SPLINE
SPL {X  -165.650, Y  +484.445, Z    +0.000, E1   +32.277, E3 +500064.677}
SPL {X  -165.650, Y  +481.524, Z    +0.000, E1   +31.089, E3 +500082.127}
SPL {X  -165.650, Y  +478.014, Z    +0.000, E1   +30.826, E3 +500095.735}
SPL {X  -165.650, Y  +474.473, Z    +0.000, E1   +30.943, E3 +500107.059}
SPL {X  -165.650, Y  +471.826, Z    +0.000, E1   +30.770, E3 +500117.243}
SPL {X  -165.650, Y  +467.753, Z    +0.000, E1   +30.878, E3 +500130.616}
SPL {X  -165.650, Y  +463.837, Z    +0.000, E1   +30.924, E3 +500143.550}
SPL {X  -165.650, Y  +461.106, Z    +0.000, E1   +30.916, E3 +500152.937}
SPL {X  -165.650, Y  +458.435, Z    +0.000, E1   +30.759, E3 +500163.145}
SPL {X  -165.650, Y  +454.220, Z    +0.000, E1   +30.954, E3 +500176.378}
SPL {X  -165.650, Y  +450.433, Z    +0.000, E1   +30.789, E3 +500190.343}
SPL {X  -165.650, Y  +447.097, Z    +0.000, E1   +30.843, E3 +500201.392}
SPL {X  -165.650, Y  +443.673, Z    +0.000, E1   +30.907, E3 +500212.699}
SPL {X  -165.650, Y  +440.976, Z    +0.000, E1   +30.719, E3 +500223.156}
SPL {X  -165.650, Y  +436.324, Z    +0.000, E1   +30.994, E3 +500237.442}
SPL {X  -165.650, Y  +432.765, Z    +0.000, E1   +30.831, E3 +500250.442}
SPL {X  -165.650, Y  +429.309, Z    +0.000, E1   +30.920, E3 +500261.783}
SPL {X  -165.650, Y  +424.918, Z    +0.000, E1   +30.862, E3 +500277.240}
SPL {X  -165.650, Y  +421.437, Z    +0.000, E1   +30.833, E3 +500289.209}
SPL {X  -165.650, Y  +417.366, Z    +0.000, E1   +30.879, E3 +500303.049}
SPL {X  -165.650, Y  +413.181, Z    +0.000, E1   +30.815, E3 +500317.647}
SPL {X  -165.650, Y  +408.547, Z    +0.000, E1   +30.964, E3 +500332.649}
SPL {X  -165.650, Y  +403.421, Z    +0.000, E1   +30.863, E3 +500350.867}
SPL {X  -165.650, Y  +398.147, Z    +0.000, E1   +30.902, E3 +500368.628}
SPL {X  -165.650, Y  +394.694, Z    +0.000, E1   +30.805, E3 +500380.936}
SPL {X  -165.650, Y  +391.522, Z    +0.000, E1   +30.837, E3 +500391.617}
SPL {X  -165.650, Y  +387.533, Z    +0.000, E1   +30.858, E3 +500405.243}
SPL {X  -165.650, Y  +383.627, Z    +0.000, E1   +30.885, E3 +500418.303}
SPL {X  -165.650, Y  +379.886, Z    +0.000, E1   +30.887, E3 +500431.192}
SPL {X  -165.614, Y  +375.058, Z    +0.000, E1   +30.905, E3 +500447.645}
SPL {X  -165.492, Y  +371.263, Z    +0.000, E1   +30.913, E3 +500460.359}
SPL {X  -165.379, Y  +369.027, Z    +0.000, E1   +30.727, E3 +500469.297}
SPL {X  -165.167, Y  +365.866, Z    +0.000, E1   +30.741, E3 +500480.071}
SPL {X  -164.892, Y  +362.671, Z    +0.000, E1   +30.830, E3 +500490.395}
SPL {X  -164.570, Y  +359.612, Z    +0.000, E1   +30.773, E3 +500501.208}
SPL {X  -164.104, Y  +355.923, Z    +0.000, E1   +30.626, E3 +500514.924}
SPL {X  -163.573, Y  +352.353, Z    +0.000, E1   +30.451, E3 +500528.189}
SPL {X  -162.476, Y  +346.230, Z    +0.000, E1   +31.677, E3 +500540.770}
SPL {X  -152.976, Y  +314.952, Z    +0.000, E1   +38.607, E3 +500589.735}
SPL {X  -137.967, Y  +286.821, Z    +0.000, E1   +43.969, E3 +500632.956}
ENDSPLINE

SPLINE
SPL {X  -153.316, Y  +315.777, Z    +0.000, E1   +33.140, E3 +500675.584}
SPL {X  -164.446, Y  +358.564, Z    +0.000, E1   +15.149, E3 +500640.795}
SPL {X  -165.510, Y  +371.680, Z    +0.000, E1    +7.684, E3 +500644.850}
SPL {X  -165.628, Y  +375.818, Z    +0.000, E1    +5.016, E3 +500652.780}
SPL {X  -165.650, Y  +383.362, Z    +0.000, E1    +0.177, E3 +500633.813}
SPL {X  -165.650, Y  +383.923, Z    +0.000, E1    -0.215, E3 +500646.971}
SPL {X  -165.650, Y  +388.083, Z    +0.000, E1    -3.355, E3 +500645.834}
SPL {X  -165.650, Y  +395.510, Z    +0.000, E1    -9.810, E3 +500641.960}
SPL {X  -165.650, Y  +403.066, Z    +0.000, E1   -17.886, E3 +500634.793}
SPL {X  -165.650, Y  +414.811, Z    +0.000, E1   -28.314, E3 +500636.275}
SPL {X  -165.650, Y  +423.479, Z    +0.000, E1   -29.012, E3 +500660.203}
SPL {X  -165.650, Y  +435.050, Z    +0.000, E1   -34.610, E3 +500668.538}
SPL {X  -165.650, Y  +446.725, Z    +0.000, E1   -39.593, E3 +500674.799}
SPL {X  -165.650, Y  +462.890, Z    +0.000, E1   -40.484, E3 +500705.975}
ENDSPLINE

SPLINE
SPL {X  -165.650, Y  +446.920, Z    +0.000, E1   -31.238, E3 +500718.301}
ENDSPLINE

SPLINE
SPL {X  -165.650, Y  +447.935, Z    +0.000, E1   -30.213, E3 +500728.589}
SPL {X  -165.650, Y  +451.020, Z    +0.000, E1   -30.224, E3 +500739.409}
SPL {X  -165.650, Y  +454.519, Z    +0.000, E1   -30.374, E3 +500750.592}
SPL {X  -165.650, Y  +457.429, Z    +0.000, E1   -30.029, E3 +500763.293}
SPL {X  -165.650, Y  +461.678, Z    +0.000, E1   -30.426, E3 +500775.418}
SPL {X  -165.650, Y  +463.853, Z    +0.000, E1   -30.103, E3 +500785.258}
SPL {X  -165.650, Y  +468.397, Z    +0.000, E1   -30.302, E3 +500800.061}
SPL {X  -165.650, Y  +472.566, Z    +0.000, E1   -30.124, E3 +500815.771}
SPL {X  -165.650, Y  +475.265, Z    +0.000, E1   -30.034, E3 +500825.808}
SPL {X  -165.650, Y  +477.862, Z    +0.000, E1   -30.319, E3 +500833.000}
SPL {X  -165.650, Y  +481.042, Z    +0.000, E1   -30.192, E3 +500845.260}
SPL {X  -165.650, Y  +485.236, Z    +0.000, E1   -30.294, E3 +500859.116}
SPL {X  -165.650, Y  +488.041, Z    +0.000, E1   -30.253, E3 +500869.237}
SPL {X  -165.650, Y  +491.281, Z    +0.000, E1   -30.148, E3 +500881.375}
SPL {X  -165.650, Y  +495.051, Z    +0.000, E1   -30.213, E3 +500894.184}
SPL {X  -165.650, Y  +499.546, Z    +0.000, E1   -30.283, E3 +500909.627}
SPL {X  -165.650, Y  +503.544, Z    +0.000, E1   -30.247, E3 +500923.695}
SPL {X  -165.650, Y  +506.344, Z    +0.000, E1   -30.129, E3 +500934.364}
SPL {X  -165.650, Y  +509.866, Z    +0.000, E1   -30.236, E3 +500946.033}
SPL {X  -165.650, Y  +513.685, Z    +0.000, E1   -30.234, E3 +500959.529}
SPL {X  -165.650, Y  +517.919, Z    +0.000, E1   -30.227, E3 +500974.436}
SPL {X  -165.650, Y  +521.521, Z    +0.000, E1   -30.210, E3 +500987.111}
SPL {X  -165.650, Y  +525.344, Z    +0.000, E1   -30.269, E3 +501000.217}
SPL {X  -165.650, Y  +528.152, Z    +0.000, E1   -29.991, E3 +501011.858}
SPL {X  -165.650, Y  +531.783, Z    +0.000, E1   -30.416, E3 +501021.751}
SPL {X  -165.650, Y  +534.115, Z    +0.000, E1   -30.089, E3 +501032.133}
SPL {X  -165.650, Y  +537.522, Z    +0.000, E1   -30.251, E3 +501043.047}
SPL {X  -165.650, Y  +540.621, Z    +0.000, E1   -30.014, E3 +501055.608}
SPL {X  -165.650, Y  +544.944, Z    +0.000, E1   -30.447, E3 +501067.808}
SPL {X  -165.650, Y  +547.199, Z    +0.000, E1   -30.132, E3 +501077.782}
SPL {X  -165.650, Y  +550.512, Z    +0.000, E1   -30.197, E3 +501089.107}
SPL {X  -165.650, Y  +553.852, Z    +0.000, E1   -30.156, E3 +501101.048}
SPL {X  -165.650, Y  +557.277, Z    +0.000, E1   -30.150, E3 +501113.223}
SPL {X  -165.650, Y  +561.168, Z    +0.000, E1   -30.194, E3 +501126.604}
SPL {X  -165.650, Y  +565.528, Z    +0.000, E1   -30.192, E3 +501142.087}
SPL {X  -165.650, Y  +570.048, Z    +0.000, E1   -30.238, E3 +501157.518}
SPL {X  -165.650, Y  +573.110, Z    +0.000, E1   -30.057, E3 +501169.503}
SPL {X  -165.650, Y  +577.587, Z    +0.000, E1   -30.270, E3 +501183.942}
SPL {X  -165.650, Y  +581.190, Z    +0.000, E1   -30.107, E3 +501197.581}
SPL {X  -165.650, Y  +585.053, Z    +0.000, E1   -30.090, E3 +501211.451}
ENDSPLINE

SPLINE
SPL {X  -165.650, Y  +484.445, Z    +0.000, E1   +32.277, E3 +501228.856}
SPL {X  -165.650, Y  +481.524, Z    +0.000, E1   +31.089, E3 +501246.306}
SPL {X  -165.650, Y  +478.014, Z    +0.000, E1   +30.826, E3 +501259.914}
SPL {X  -165.650, Y  +474.473, Z    +0.000, E1   +30.943, E3 +501271.238}
SPL {X  -165.650, Y  +471.826, Z    +0.000, E1   +30.770, E3 +501281.422}
SPL {X  -165.650, Y  +467.753, Z    +0.000, E1   +30.878, E3 +501294.795}
SPL {X  -165.650, Y  +463.837, Z    +0.000, E1   +30.924, E3 +501307.729}
SPL {X  -165.650, Y  +461.106, Z    +0.000, E1   +30.916, E3 +501317.116}
SPL {X  -165.650, Y  +458.435, Z    +0.000, E1   +30.759, E3 +501327.324}
SPL {X  -165.650, Y  +454.220, Z    +0.000, E1   +30.954, E3 +501340.557}
SPL {X  -165.650, Y  +450.433, Z    +0.000, E1   +30.789, E3 +501354.522}
SPL {X  -165.650, Y  +447.097, Z    +0.000, E1   +30.843, E3 +501365.571}
SPL {X  -165.650, Y  +443.673, Z    +0.000, E1   +30.907, E3 +501376.878}
SPL {X  -165.650, Y  +440.976, Z    +0.000, E1   +30.719, E3 +501387.335}
SPL {X  -165.650, Y  +436.324, Z    +0.000, E1   +30.994, E3 +501401.621}
SPL {X  -165.650, Y  +432.765, Z    +0.000, E1   +30.831, E3 +501414.621}
SPL {X  -165.650, Y  +429.309, Z    +0.000, E1   +30.920, E3 +501425.962}
SPL {X  -165.650, Y  +424.918, Z    +0.000, E1   +30.862, E3 +501441.419}
SPL {X  -165.650, Y  +421.437, Z    +0.000, E1   +30.833, E3 +501453.388}
SPL {X  -165.650, Y  +418.489, Z    +0.000, E1   +30.835, E3 +501463.504}
SPL {X  -165.650, Y  +414.127, Z    +0.000, E1   +30.869, E3 +501478.413}
SPL {X  -165.650, Y  +408.547, Z    +0.000, E1   +30.964, E3 +501496.829}
SPL {X  -165.650, Y  +405.433, Z    +0.000, E1   +30.730, E3 +501508.806}
SPL {X  -165.650, Y  +401.473, Z    +0.000, E1   +30.933, E3 +501521.254}
SPL {X  -165.650, Y  +396.018, Z    +0.000, E1   +30.861, E3 +501540.439}
SPL {X  -165.650, Y  +391.522, Z    +0.000, E1   +30.837, E3 +501555.796}
SPL {X  -165.650, Y  +387.533, Z    +0.000, E1   +30.858, E3 +501569.422}
SPL {X  -165.650, Y  +383.627, Z    +0.000, E1   +30.885, E3 +501582.483}
SPL {X  -165.650, Y  +380.752, Z    +0.000, E1   +30.927, E3 +501591.996}
SPL {X  -165.648, Y  +377.739, Z    +0.000, E1   +30.835, E3 +501603.006}
SPL {X  -165.594, Y  +374.183, Z    +0.000, E1   +30.878, E3 +501614.843}
SPL {X  -165.429, Y  +369.945, Z    +0.000, E1   +30.850, E3 +501629.718}
SPL {X  -165.167, Y  +365.866, Z    +0.000, E1   +30.741, E3 +501644.250}
SPL {X  -164.892, Y  +362.671, Z    +0.000, E1   +30.830, E3 +501654.574}
SPL {X  -164.570, Y  +359.612, Z    +0.000, E1   +30.773, E3 +501665.387}
SPL {X  -164.104, Y  +355.923, Z    +0.000, E1   +30.626, E3 +501679.104}
SPL {X  -163.573, Y  +352.353, Z    +0.000, E1   +30.451, E3 +501692.368}
SPL {X  -162.976, Y  +348.856, Z    +0.000, E1   +30.757, E3 +501702.292}
SPL {X  -161.497, Y  +341.640, Z    +0.000, E1   +33.276, E3 +501709.570}
SPL {X  -152.976, Y  +314.952, Z    +0.000, E1   +38.607, E3 +501753.914}
SPL {X  -137.967, Y  +286.821, Z    +0.000, E1   +43.969, E3 +501797.135}
ENDSPLINE

SPLINE
SPL {X  -149.143, Y  +306.414, Z    +0.000, E1   +36.361, E3 +501848.268}
SPL {X  -164.268, Y  +357.145, Z    +0.000, E1   +15.880, E3 +501806.027}
SPL {X  -165.510, Y  +371.680, Z    +0.000, E1    +7.684, E3 +501809.029}
SPL {X  -165.628, Y  +375.818, Z    +0.000, E1    +5.016, E3 +501816.959}
SPL {X  -165.650, Y  +383.362, Z    +0.000, E1    +0.177, E3 +501797.992}
SPL {X  -165.650, Y  +383.923, Z    +0.000, E1    -0.215, E3 +501811.150}
SPL {X  -165.650, Y  +388.083, Z    +0.000, E1    -3.355, E3 +501810.013}
SPL {X  -165.650, Y  +395.510, Z    +0.000, E1    -9.810, E3 +501806.139}
SPL {X  -165.650, Y  +403.066, Z    +0.000, E1   -17.886, E3 +501798.973}
SPL {X  -165.650, Y  +416.345, Z    +0.000, E1   -29.511, E3 +501800.715}
SPL {X  -165.650, Y  +422.331, Z    +0.000, E1   -27.760, E3 +501826.214}
SPL {X  -165.650, Y  +441.276, Z    +0.000, E1   -37.343, E3 +501836.071}
SPL {X  -165.650, Y  +462.890, Z    +0.000, E1   -40.484, E3 +501870.154}
ENDSPLINE

SPLINE
SPL {X  -165.650, Y  +446.920, Z    +0.000, E1   -31.238, E3 +501882.480}
ENDSPLINE

SPLINE
SPL {X  -165.650, Y  +447.935, Z    +0.000, E1   -30.213, E3 +501892.768}
SPL {X  -165.650, Y  +451.020, Z    +0.000, E1   -30.224, E3 +501903.588}
SPL {X  -165.650, Y  +454.519, Z    +0.000, E1   -30.374, E3 +501914.771}
SPL {X  -165.650, Y  +457.429, Z    +0.000, E1   -30.029, E3 +501927.473}
SPL {X  -165.650, Y  +461.678, Z    +0.000, E1   -30.426, E3 +501939.597}
SPL {X  -165.650, Y  +463.853, Z    +0.000, E1   -30.103, E3 +501949.437}
SPL {X  -165.650, Y  +468.397, Z    +0.000, E1   -30.302, E3 +501964.241}
SPL {X  -165.650, Y  +472.566, Z    +0.000, E1   -30.124, E3 +501979.950}
SPL {X  -165.650, Y  +476.540, Z    +0.000, E1   -30.193, E3 +501993.494}
SPL {X  -165.650, Y  +481.042, Z    +0.000, E1   -30.192, E3 +502009.439}
SPL {X  -165.650, Y  +485.236, Z    +0.000, E1   -30.294, E3 +502023.295}
SPL {X  -165.650, Y  +489.057, Z    +0.000, E1   -30.341, E3 +502036.501}
SPL {X  -165.650, Y  +491.647, Z    +0.000, E1   -29.894, E3 +502048.434}
SPL {X  -165.650, Y  +495.051, Z    +0.000, E1   -30.213, E3 +502058.363}
SPL {X  -165.650, Y  +498.418, Z    +0.000, E1   -30.282, E3 +502069.656}
SPL {X  -165.650, Y  +502.421, Z    +0.000, E1   -30.263, E3 +502084.013}
SPL {X  -165.650, Y  +506.344, Z    +0.000, E1   -30.129, E3 +502098.543}
SPL {X  -165.650, Y  +509.866, Z    +0.000, E1   -30.236, E3 +502110.212}
SPL {X  -165.650, Y  +513.685, Z    +0.000, E1   -30.234, E3 +502123.709}
SPL {X  -165.650, Y  +517.919, Z    +0.000, E1   -30.227, E3 +502138.615}
SPL {X  -165.650, Y  +521.521, Z    +0.000, E1   -30.210, E3 +502151.290}
SPL {X  -165.650, Y  +525.344, Z    +0.000, E1   -30.269, E3 +502164.396}
SPL {X  -165.650, Y  +528.152, Z    +0.000, E1   -29.991, E3 +502176.037}
SPL {X  -165.650, Y  +531.783, Z    +0.000, E1   -30.416, E3 +502185.930}
SPL {X  -165.650, Y  +534.115, Z    +0.000, E1   -30.089, E3 +502196.312}
SPL {X  -165.650, Y  +537.522, Z    +0.000, E1   -30.251, E3 +502207.227}
SPL {X  -165.650, Y  +540.621, Z    +0.000, E1   -30.014, E3 +502219.787}
SPL {X  -165.650, Y  +544.944, Z    +0.000, E1   -30.447, E3 +502231.987}
SPL {X  -165.650, Y  +548.549, Z    +0.000, E1   -30.216, E3 +502246.311}
SPL {X  -165.650, Y  +553.092, Z    +0.000, E1   -30.157, E3 +502262.653}
SPL {X  -165.650, Y  +556.274, Z    +0.000, E1   -30.127, E3 +502273.908}
SPL {X  -165.650, Y  +560.243, Z    +0.000, E1   -30.214, E3 +502287.574}
SPL {X  -165.650, Y  +565.528, Z    +0.000, E1   -30.192, E3 +502306.266}
SPL {X  -165.650, Y  +570.048, Z    +0.000, E1   -30.238, E3 +502321.697}
SPL {X  -165.650, Y  +573.110, Z    +0.000, E1   -30.057, E3 +502333.682}
SPL {X  -165.650, Y  +577.587, Z    +0.000, E1   -30.270, E3 +502348.121}
SPL {X  -165.650, Y  +581.190, Z    +0.000, E1   -30.107, E3 +502361.760}
SPL {X  -165.650, Y  +585.053, Z    +0.000, E1   -30.090, E3 +502375.631}
ENDSPLINE

SPLINE
SPL {X  -165.650, Y  +484.445, Z    +0.000, E1   +32.277, E3 +502393.035}
SPL {X  -165.650, Y  +481.524, Z    +0.000, E1   +31.089, E3 +502410.486}
SPL {X  -165.650, Y  +478.014, Z    +0.000, E1   +30.826, E3 +502424.093}
SPL {X  -165.650, Y  +474.473, Z    +0.000, E1   +30.943, E3 +502435.418}
SPL {X  -165.650, Y  +471.826, Z    +0.000, E1   +30.770, E3 +502445.601}
SPL {X  -165.650, Y  +467.753, Z    +0.000, E1   +30.878, E3 +502458.974}
SPL {X  -165.650, Y  +463.837, Z    +0.000, E1   +30.924, E3 +502471.908}
SPL {X  -165.650, Y  +461.106, Z    +0.000, E1   +30.916, E3 +502481.295}
SPL {X  -165.650, Y  +458.435, Z    +0.000, E1   +30.759, E3 +502491.503}
SPL {X  -165.650, Y  +454.220, Z    +0.000, E1   +30.954, E3 +502504.736}
SPL {X  -165.650, Y  +450.433, Z    +0.000, E1   +30.789, E3 +502518.701}
SPL {X  -165.650, Y  +447.097, Z    +0.000, E1   +30.843, E3 +502529.750}
SPL {X  -165.650, Y  +443.673, Z    +0.000, E1   +30.907, E3 +502541.057}
SPL {X  -165.650, Y  +440.976, Z    +0.000, E1   +30.719, E3 +502551.514}
SPL {X  -165.650, Y  +436.324, Z    +0.000, E1   +30.994, E3 +502565.800}
SPL {X  -165.650, Y  +432.765, Z    +0.000, E1   +30.831, E3 +502578.800}
SPL {X  -165.650, Y  +429.309, Z    +0.000, E1   +30.920, E3 +502590.141}
SPL {X  -165.650, Y  +424.918, Z    +0.000, E1   +30.862, E3 +502605.598}
SPL {X  -165.650, Y  +421.437, Z    +0.000, E1   +30.833, E3 +502617.567}
SPL {X  -165.650, Y  +417.366, Z    +0.000, E1   +30.879, E3 +502631.407}
SPL {X  -165.650, Y  +413.181, Z    +0.000, E1   +30.815, E3 +502646.005}
SPL {X  -165.650, Y  +408.547, Z    +0.000, E1   +30.964, E3 +502661.008}
SPL {X  -165.650, Y  +403.421, Z    +0.000, E1   +30.863, E3 +502679.225}
SPL {X  -165.650, Y  +398.147, Z    +0.000, E1   +30.902, E3 +502696.986}
SPL {X  -165.650, Y  +394.694, Z    +0.000, E1   +30.805, E3 +502709.294}
SPL {X  -165.650, Y  +391.522, Z    +0.000, E1   +30.837, E3 +502719.975}
SPL {X  -165.650, Y  +387.533, Z    +0.000, E1   +30.858, E3 +502733.601}
SPL {X  -165.650, Y  +383.627, Z    +0.000, E1   +30.885, E3 +502746.662}
SPL {X  -165.650, Y  +379.886, Z    +0.000, E1   +30.887, E3 +502759.550}
SPL {X  -165.614, Y  +375.058, Z    +0.000, E1   +30.905, E3 +502776.003}
SPL {X  -165.492, Y  +371.263, Z    +0.000, E1   +30.913, E3 +502788.717}
SPL {X  -165.379, Y  +369.027, Z    +0.000, E1   +30.727, E3 +502797.655}
SPL {X  -165.167, Y  +365.866, Z    +0.000, E1   +30.741, E3 +502808.429}
SPL {X  -164.892, Y  +362.671, Z    +0.000, E1   +30.830, E3 +502818.754}
SPL {X  -164.570, Y  +359.612, Z    +0.000, E1   +30.773, E3 +502829.566}
SPL {X  -164.104, Y  +355.923, Z    +0.000, E1   +30.626, E3 +502843.283}
SPL {X  -163.573, Y  +352.353, Z    +0.000, E1   +30.451, E3 +502856.547}
SPL {X  -162.476, Y  +346.230, Z    +0.000, E1   +31.677, E3 +502869.128}
SPL {X  -152.976, Y  +314.952, Z    +0.000, E1   +38.607, E3 +502918.093}
SPL {X  -137.967, Y  +286.821, Z    +0.000, E1   +43.969, E3 +502961.315}
ENDSPLINE

SPLINE
SPL {X  -153.316, Y  +315.777, Z    +0.000, E1   +33.140, E3 +503003.942}
SPL {X  -164.446, Y  +358.564, Z    +0.000, E1   +15.149, E3 +502969.153}
SPL {X  -165.379, Y  +369.025, Z    +0.000, E1    +9.158, E3 +502974.878}
SPL {X  -165.612, Y  +374.969, Z    +0.000, E1    +5.630, E3 +502977.553}
SPL {X  -165.650, Y  +383.362, Z    +0.000, E1    +0.177, E3 +502962.172}
SPL {X  -165.650, Y  +383.923, Z    +0.000, E1    -0.215, E3 +502975.329}
SPL {X  -165.650, Y  +388.083, Z    +0.000, E1    -3.355, E3 +502974.192}
SPL {X  -165.650, Y  +395.510, Z    +0.000, E1    -9.810, E3 +502970.318}
SPL {X  -165.650, Y  +403.066, Z    +0.000, E1   -17.886, E3 +502963.152}
SPL {X  -165.650, Y  +414.811, Z    +0.000, E1   -28.314, E3 +502964.633}
SPL {X  -165.650, Y  +423.479, Z    +0.000, E1   -29.012, E3 +502988.562}
SPL {X  -165.650, Y  +441.276, Z    +0.000, E1   -37.343, E3 +503000.250}
SPL {X  -165.650, Y  +462.890, Z    +0.000, E1   -40.484, E3 +503034.333}
ENDSPLINE

SPLINE
SPL {X  -165.650, Y  +446.920, Z    +0.000, E1   -31.238, E3 +503046.659}
ENDSPLINE

SPLINE
SPL {X  -165.650, Y  +447.935, Z    +0.000, E1   -30.213, E3 +503056.947}
SPL {X  -165.650, Y  +451.020, Z    +0.000, E1   -30.224, E3 +503067.768}
SPL {X  -165.650, Y  +454.519, Z    +0.000, E1   -30.374, E3 +503078.950}
SPL {X  -165.650, Y  +457.429, Z    +0.000, E1   -30.029, E3 +503091.652}
SPL {X  -165.650, Y  +461.678, Z    +0.000, E1   -30.426, E3 +503103.776}
SPL {X  -165.650, Y  +463.853, Z    +0.000, E1   -30.103, E3 +503113.616}
SPL {X  -165.650, Y  +468.397, Z    +0.000, E1   -30.302, E3 +503128.420}
SPL {X  -165.650, Y  +472.566, Z    +0.000, E1   -30.124, E3 +503144.129}
SPL {X  -165.650, Y  +476.540, Z    +0.000, E1   -30.193, E3 +503157.673}
SPL {X  -165.650, Y  +481.042, Z    +0.000, E1   -30.192, E3 +503173.618}
SPL {X  -165.650, Y  +485.236, Z    +0.000, E1   -30.294, E3 +503187.474}
SPL {X  -165.650, Y  +489.057, Z    +0.000, E1   -30.341, E3 +503200.680}
SPL {X  -165.650, Y  +491.647, Z    +0.000, E1   -29.894, E3 +503212.613}
SPL {X  -165.650, Y  +495.051, Z    +0.000, E1   -30.213, E3 +503222.542}
SPL {X  -165.650, Y  +499.546, Z    +0.000, E1   -30.283, E3 +503237.985}
SPL {X  -165.650, Y  +503.544, Z    +0.000, E1   -30.247, E3 +503252.053}
SPL {X  -165.650, Y  +506.344, Z    +0.000, E1   -30.129, E3 +503262.722}
SPL {X  -165.650, Y  +510.660, Z    +0.000, E1   -30.223, E3 +503277.425}
SPL {X  -165.650, Y  +514.670, Z    +0.000, E1   -30.278, E3 +503290.935}
SPL {X  -165.650, Y  +517.919, Z    +0.000, E1   -30.227, E3 +503302.795}
SPL {X  -165.650, Y  +522.822, Z    +0.000, E1   -30.289, E3 +503319.684}
SPL {X  -165.650, Y  +527.393, Z    +0.000, E1   -30.104, E3 +503336.932}
SPL {X  -165.650, Y  +531.783, Z    +0.000, E1   -30.416, E3 +503350.109}
SPL {X  -165.650, Y  +534.115, Z    +0.000, E1   -30.089, E3 +503360.491}
SPL {X  -165.650, Y  +538.363, Z    +0.000, E1   -30.232, E3 +503374.661}
SPL {X  -165.650, Y  +543.650, Z    +0.000, E1   -30.281, E3 +503392.881}
SPL {X  -165.650, Y  +548.549, Z    +0.000, E1   -30.216, E3 +503410.490}
SPL {X  -165.650, Y  +553.092, Z    +0.000, E1   -30.157, E3 +503426.832}
SPL {X  -165.650, Y  +556.274, Z    +0.000, E1   -30.127, E3 +503438.087}
SPL {X  -165.650, Y  +560.243, Z    +0.000, E1   -30.214, E3 +503451.753}
SPL {X  -165.650, Y  +565.528, Z    +0.000, E1   -30.192, E3 +503470.445}
SPL {X  -165.650, Y  +570.048, Z    +0.000, E1   -30.238, E3 +503485.876}
SPL {X  -165.650, Y  +573.110, Z    +0.000, E1   -30.057, E3 +503497.861}
SPL {X  -165.650, Y  +577.587, Z    +0.000, E1   -30.270, E3 +503512.300}
SPL {X  -165.650, Y  +581.190, Z    +0.000, E1   -30.107, E3 +503525.939}
SPL {X  -165.650, Y  +585.053, Z    +0.000, E1   -30.090, E3 +503539.810}
ENDSPLINE

SPLINE
SPL {X  -165.650, Y  +484.445, Z    +0.000, E1   +32.277, E3 +503557.214}
SPL {X  -165.650, Y  +481.524, Z    +0.000, E1   +31.089, E3 +503574.665}
SPL {X  -165.650, Y  +478.014, Z    +0.000, E1   +30.826, E3 +503588.272}
SPL {X  -165.650, Y  +474.473, Z    +0.000, E1   +30.943, E3 +503599.597}
SPL {X  -165.650, Y  +471.826, Z    +0.000, E1   +30.770, E3 +503609.780}
SPL {X  -165.650, Y  +467.753, Z    +0.000, E1   +30.878, E3 +503623.154}
SPL {X  -165.650, Y  +463.837, Z    +0.000, E1   +30.924, E3 +503636.087}
SPL {X  -165.650, Y  +461.106, Z    +0.000, E1   +30.916, E3 +503645.474}
SPL {X  -165.650, Y  +457.156, Z    +0.000, E1   +30.860, E3 +503659.551}
SPL {X  -165.650, Y  +453.156, Z    +0.000, E1   +30.934, E3 +503672.525}
SPL {X  -165.650, Y  +450.433, Z    +0.000, E1   +30.789, E3 +503682.880}
SPL {X  -165.650, Y  +447.097, Z    +0.000, E1   +30.843, E3 +503693.929}
SPL {X  -165.650, Y  +443.673, Z    +0.000, E1   +30.907, E3 +503705.236}
SPL {X  -165.650, Y  +439.486, Z    +0.000, E1   +30.857, E3 +503720.046}
SPL {X  -165.650, Y  +435.146, Z    +0.000, E1   +30.969, E3 +503733.965}
SPL {X  -165.650, Y  +431.607, Z    +0.000, E1   +30.889, E3 +503746.680}
SPL {X  -165.650, Y  +427.340, Z    +0.000, E1   +30.870, E3 +503761.391}
SPL {X  -165.650, Y  +423.901, Z    +0.000, E1   +30.858, E3 +503773.148}
SPL {X  -165.650, Y  +421.437, Z    +0.000, E1   +30.833, E3 +503781.746}
SPL {X  -165.650, Y  +418.489, Z    +0.000, E1   +30.835, E3 +503791.863}
SPL {X  -165.650, Y  +414.127, Z    +0.000, E1   +30.869, E3 +503806.771}
SPL {X  -165.650, Y  +408.547, Z    +0.000, E1   +30.964, E3 +503825.187}
SPL {X  -165.650, Y  +405.433, Z    +0.000, E1   +30.730, E3 +503837.164}
SPL {X  -165.650, Y  +401.473, Z    +0.000, E1   +30.933, E3 +503849.612}
SPL {X  -165.650, Y  +396.018, Z    +0.000, E1   +30.861, E3 +503868.797}
SPL {X  -165.650, Y  +391.522, Z    +0.000, E1   +30.837, E3 +503884.154}
SPL {X  -165.650, Y  +387.533, Z    +0.000, E1   +30.858, E3 +503897.780}
SPL {X  -165.650, Y  +383.627, Z    +0.000, E1   +30.885, E3 +503910.841}
SPL {X  -165.650, Y  +380.752, Z    +0.000, E1   +30.927, E3 +503920.355}
SPL {X  -165.648, Y  +377.739, Z    +0.000, E1   +30.835, E3 +503931.364}
SPL {X  -165.594, Y  +374.183, Z    +0.000, E1   +30.878, E3 +503943.201}
SPL {X  -165.429, Y  +369.945, Z    +0.000, E1   +30.850, E3 +503958.076}
SPL {X  -165.167, Y  +365.866, Z    +0.000, E1   +30.741, E3 +503972.609}
SPL {X  -164.892, Y  +362.671, Z    +0.000, E1   +30.830, E3 +503982.933}
SPL {X  -164.570, Y  +359.612, Z    +0.000, E1   +30.773, E3 +503993.745}
SPL {X  -164.104, Y  +355.923, Z    +0.000, E1   +30.626, E3 +504007.462}
SPL {X  -163.573, Y  +352.353, Z    +0.000, E1   +30.451, E3 +504020.727}
SPL {X  -162.976, Y  +348.856, Z    +0.000, E1   +30.757, E3 +504030.650}
SPL {X  -161.497, Y  +341.640, Z    +0.000, E1   +33.276, E3 +504037.928}
SPL {X  -152.976, Y  +314.952, Z    +0.000, E1   +38.607, E3 +504082.272}
SPL {X  -137.967, Y  +286.821, Z    +0.000, E1   +43.969, E3 +504125.494}
ENDSPLINE

SPLINE
SPL {X  -149.143, Y  +306.414, Z    +0.000, E1   +36.361, E3 +504176.626}
SPL {X  -164.268, Y  +357.145, Z    +0.000, E1   +15.880, E3 +504134.385}
SPL {X  -165.510, Y  +371.680, Z    +0.000, E1    +7.684, E3 +504137.388}
SPL {X  -165.628, Y  +375.818, Z    +0.000, E1    +5.016, E3 +504145.317}
SPL {X  -165.650, Y  +383.362, Z    +0.000, E1    +0.177, E3 +504126.351}
SPL {X  -165.650, Y  +383.923, Z    +0.000, E1    -0.215, E3 +504139.508}
SPL {X  -165.650, Y  +388.083, Z    +0.000, E1    -3.355, E3 +504138.371}
SPL {X  -165.650, Y  +395.510, Z    +0.000, E1    -9.810, E3 +504134.498}
SPL {X  -165.650, Y  +403.066, Z    +0.000, E1   -17.886, E3 +504127.331}
SPL {X  -165.650, Y  +416.345, Z    +0.000, E1   -29.511, E3 +504129.073}
SPL {X  -165.650, Y  +422.331, Z    +0.000, E1   -27.760, E3 +504154.572}
SPL {X  -165.650, Y  +441.276, Z    +0.000, E1   -37.343, E3 +504164.430}
SPL {X  -165.650, Y  +462.890, Z    +0.000, E1   -40.484, E3 +504198.512}
ENDSPLINE

SPLINE
SPL {X  -165.650, Y  +446.920, Z    +0.000, E1   -31.238, E3 +504210.838}
ENDSPLINE

SPLINE
SPL {X  -165.650, Y  +447.935, Z    +0.000, E1   -30.213, E3 +504221.126}
SPL {X  -165.650, Y  +451.020, Z    +0.000, E1   -30.224, E3 +504231.947}
SPL {X  -165.650, Y  +454.519, Z    +0.000, E1   -30.374, E3 +504243.129}
SPL {X  -165.650, Y  +457.429, Z    +0.000, E1   -30.029, E3 +504255.831}
SPL {X  -165.650, Y  +461.678, Z    +0.000, E1   -30.426, E3 +504267.955}
SPL {X  -165.650, Y  +463.853, Z    +0.000, E1   -30.103, E3 +504277.795}
SPL {X  -165.650, Y  +468.397, Z    +0.000, E1   -30.302, E3 +504292.599}
SPL {X  -165.650, Y  +472.566, Z    +0.000, E1   -30.124, E3 +504308.308}
SPL {X  -165.650, Y  +476.540, Z    +0.000, E1   -30.193, E3 +504321.852}
SPL {X  -165.650, Y  +481.042, Z    +0.000, E1   -30.192, E3 +504337.797}
SPL {X  -165.650, Y  +485.236, Z    +0.000, E1   -30.294, E3 +504351.653}
SPL {X  -165.650, Y  +489.057, Z    +0.000, E1   -30.341, E3 +504364.859}
SPL {X  -165.650, Y  +491.647, Z    +0.000, E1   -29.894, E3 +504376.792}
SPL {X  -165.650, Y  +495.051, Z    +0.000, E1   -30.213, E3 +504386.721}
SPL {X  -165.650, Y  +498.418, Z    +0.000, E1   -30.282, E3 +504398.014}
SPL {X  -165.650, Y  +502.421, Z    +0.000, E1   -30.263, E3 +504412.371}
SPL {X  -165.650, Y  +506.344, Z    +0.000, E1   -30.129, E3 +504426.901}
SPL {X  -165.650, Y  +509.866, Z    +0.000, E1   -30.236, E3 +504438.570}
SPL {X  -165.650, Y  +513.685, Z    +0.000, E1   -30.234, E3 +504452.067}
SPL {X  -165.650, Y  +517.919, Z    +0.000, E1   -30.227, E3 +504466.974}
SPL {X  -165.650, Y  +521.521, Z    +0.000, E1   -30.210, E3 +504479.648}
SPL {X  -165.650, Y  +525.344, Z    +0.000, E1   -30.269, E3 +504492.755}
SPL {X  -165.650, Y  +528.152, Z    +0.000, E1   -29.991, E3 +504504.396}
SPL {X  -165.650, Y  +531.783, Z    +0.000, E1   -30.416, E3 +504514.288}
SPL {X  -165.650, Y  +534.115, Z    +0.000, E1   -30.089, E3 +504524.670}
SPL {X  -165.650, Y  +537.522, Z    +0.000, E1   -30.251, E3 +504535.585}
SPL {X  -165.650, Y  +540.621, Z    +0.000, E1   -30.014, E3 +504548.146}
SPL {X  -165.650, Y  +544.944, Z    +0.000, E1   -30.447, E3 +504560.345}
SPL {X  -165.650, Y  +548.549, Z    +0.000, E1   -30.216, E3 +504574.669}
SPL {X  -165.650, Y  +553.092, Z    +0.000, E1   -30.157, E3 +504591.011}
SPL {X  -165.650, Y  +556.274, Z    +0.000, E1   -30.127, E3 +504602.266}
SPL {X  -165.650, Y  +560.243, Z    +0.000, E1   -30.214, E3 +504615.932}
SPL {X  -165.650, Y  +565.528, Z    +0.000, E1   -30.192, E3 +504634.624}
SPL {X  -165.650, Y  +570.048, Z    +0.000, E1   -30.238, E3 +504650.055}
SPL {X  -165.650, Y  +573.110, Z    +0.000, E1   -30.057, E3 +504662.040}
SPL {X  -165.650, Y  +577.587, Z    +0.000, E1   -30.270, E3 +504676.479}
SPL {X  -165.650, Y  +581.190, Z    +0.000, E1   -30.107, E3 +504690.119}
SPL {X  -165.650, Y  +585.053, Z    +0.000, E1   -30.090, E3 +504703.989}
ENDSPLINE

SPLINE
SPL {X  -165.650, Y  +484.445, Z    +0.000, E1   +32.277, E3 +504721.393}
SPL {X  -165.650, Y  +481.524, Z    +0.000, E1   +31.089, E3 +504738.844}
SPL {X  -165.650, Y  +478.014, Z    +0.000, E1   +30.826, E3 +504752.451}
SPL {X  -165.650, Y  +474.473, Z    +0.000, E1   +30.943, E3 +504763.776}
SPL {X  -165.650, Y  +471.826, Z    +0.000, E1   +30.770, E3 +504773.959}
SPL {X  -165.650, Y  +467.753, Z    +0.000, E1   +30.878, E3 +504787.333}
SPL {X  -165.650, Y  +463.837, Z    +0.000, E1   +30.924, E3 +504800.267}
SPL {X  -165.650, Y  +461.106, Z    +0.000, E1   +30.916, E3 +504809.654}
SPL {X  -165.650, Y  +457.156, Z    +0.000, E1   +30.860, E3 +504823.730}
SPL {X  -165.650, Y  +453.156, Z    +0.000, E1   +30.934, E3 +504836.704}
SPL {X  -165.650, Y  +450.433, Z    +0.000, E1   +30.789, E3 +504847.059}
SPL {X  -165.650, Y  +447.097, Z    +0.000, E1   +30.843, E3 +504858.108}
SPL {X  -165.650, Y  +443.673, Z    +0.000, E1   +30.907, E3 +504869.415}
SPL {X  -165.650, Y  +439.486, Z    +0.000, E1   +30.857, E3 +504884.225}
SPL {X  -165.650, Y  +435.146, Z    +0.000, E1   +30.969, E3 +504898.144}
SPL {X  -165.650, Y  +431.607, Z    +0.000, E1   +30.889, E3 +504910.859}
SPL {X  -165.650, Y  +427.340, Z    +0.000, E1   +30.870, E3 +504925.571}
SPL {X  -165.650, Y  +423.901, Z    +0.000, E1   +30.858, E3 +504937.327}
SPL {X  -165.650, Y  +421.437, Z    +0.000, E1   +30.833, E3 +504945.925}
SPL {X  -165.650, Y  +418.489, Z    +0.000, E1   +30.835, E3 +504956.042}
SPL {X  -165.650, Y  +415.831, Z    +0.000, E1   +30.847, E3 +504965.004}
SPL {X  -165.650, Y  +412.139, Z    +0.000, E1   +30.870, E3 +504977.715}
SPL {X  -165.650, Y  +406.834, Z    +0.000, E1   +30.919, E3 +504995.544}
SPL {X  -165.650, Y  +402.516, Z    +0.000, E1   +30.874, E3 +505010.466}
SPL {X  -165.650, Y  +398.147, Z    +0.000, E1   +30.902, E3 +505025.344}
SPL {X  -165.650, Y  +394.694, Z    +0.000, E1   +30.805, E3 +505037.653}
SPL {X  -165.650, Y  +391.522, Z    +0.000, E1   +30.837, E3 +505048.333}
SPL {X  -165.650, Y  +387.533, Z    +0.000, E1   +30.858, E3 +505061.960}
SPL {X  -165.650, Y  +383.627, Z    +0.000, E1   +30.885, E3 +505075.020}
SPL {X  -165.650, Y  +380.752, Z    +0.000, E1   +30.927, E3 +505084.534}
SPL {X  -165.648, Y  +377.739, Z    +0.000, E1   +30.835, E3 +505095.543}
SPL {X  -165.594, Y  +374.183, Z    +0.000, E1   +30.878, E3 +505107.380}
SPL {X  -165.429, Y  +369.945, Z    +0.000, E1   +30.850, E3 +505122.255}
SPL {X  -165.167, Y  +365.866, Z    +0.000, E1   +30.741, E3 +505136.788}
SPL {X  -164.892, Y  +362.671, Z    +0.000, E1   +30.830, E3 +505147.112}
SPL {X  -164.570, Y  +359.612, Z    +0.000, E1   +30.773, E3 +505157.924}
SPL {X  -164.104, Y  +355.923, Z    +0.000, E1   +30.626, E3 +505171.641}
SPL {X  -163.573, Y  +352.353, Z    +0.000, E1   +30.451, E3 +505184.906}
SPL {X  -162.476, Y  +346.230, Z    +0.000, E1   +31.677, E3 +505197.486}
SPL {X  -152.976, Y  +314.952, Z    +0.000, E1   +38.607, E3 +505246.452}
SPL {X  -137.967, Y  +286.821, Z    +0.000, E1   +43.969, E3 +505289.673}
ENDSPLINE

SPLINE
SPL {X  -153.316, Y  +315.777, Z    +0.000, E1   +33.140, E3 +505332.300}
SPL {X  -164.446, Y  +358.564, Z    +0.000, E1   +15.149, E3 +505297.511}
SPL {X  -165.510, Y  +371.680, Z    +0.000, E1    +7.684, E3 +505301.567}
SPL {X  -165.628, Y  +375.818, Z    +0.000, E1    +5.016, E3 +505309.496}
SPL {X  -165.650, Y  +383.362, Z    +0.000, E1    +0.177, E3 +505290.530}
SPL {X  -165.650, Y  +383.923, Z    +0.000, E1    -0.215, E3 +505303.687}
SPL {X  -165.650, Y  +388.083, Z    +0.000, E1    -3.355, E3 +505302.551}
SPL {X  -165.650, Y  +393.983, Z    +0.000, E1    -8.501, E3 +505298.949}
SPL {X  -165.650, Y  +402.241, Z    +0.000, E1   -16.711, E3 +505293.461}
SPL {X  -165.650, Y  +414.811, Z    +0.000, E1   -28.314, E3 +505292.991}
SPL {X  -165.650, Y  +423.479, Z    +0.000, E1   -29.012, E3 +505316.920}
SPL {X  -165.650, Y  +435.050, Z    +0.000, E1   -34.610, E3 +505325.254}
SPL {X  -165.650, Y  +446.725, Z    +0.000, E1   -39.593, E3 +505331.515}
SPL {X  -165.650, Y  +462.890, Z    +0.000, E1   -40.484, E3 +505362.692}
ENDSPLINE

SPLINE
SPL {X  -165.650, Y  +446.920, Z    +0.000, E1   -31.238, E3 +505375.017}
ENDSPLINE

SPLINE
SPL {X  -165.650, Y  +447.935, Z    +0.000, E1   -30.213, E3 +505385.305}
SPL {X  -165.650, Y  +451.020, Z    +0.000, E1   -30.224, E3 +505396.126}
SPL {X  -165.650, Y  +454.519, Z    +0.000, E1   -30.374, E3 +505407.308}
SPL {X  -165.650, Y  +457.429, Z    +0.000, E1   -30.029, E3 +505420.010}
SPL {X  -165.650, Y  +461.678, Z    +0.000, E1   -30.426, E3 +505432.134}
SPL {X  -165.650, Y  +463.853, Z    +0.000, E1   -30.103, E3 +505441.974}
SPL {X  -165.650, Y  +468.397, Z    +0.000, E1   -30.302, E3 +505456.778}
SPL {X  -165.650, Y  +472.566, Z    +0.000, E1   -30.124, E3 +505472.487}
SPL {X  -165.650, Y  +476.540, Z    +0.000, E1   -30.193, E3 +505486.031}
SPL {X  -165.650, Y  +480.320, Z    +0.000, E1   -30.163, E3 +505499.509}
SPL {X  -165.650, Y  +484.477, Z    +0.000, E1   -30.274, E3 +505513.398}
SPL {X  -165.650, Y  +488.041, Z    +0.000, E1   -30.253, E3 +505525.954}
SPL {X  -165.650, Y  +491.281, Z    +0.000, E1   -30.148, E3 +505538.092}
SPL {X  -165.650, Y  +495.051, Z    +0.000, E1   -30.213, E3 +505550.900}
SPL {X  -165.650, Y  +498.418, Z    +0.000, E1   -30.282, E3 +505562.193}
SPL {X  -165.650, Y  +502.421, Z    +0.000, E1   -30.263, E3 +505576.551}
SPL {X  -165.650, Y  +506.344, Z    +0.000, E1   -30.129, E3 +505591.080}
SPL {X  -165.650, Y  +509.866, Z    +0.000, E1   -30.236, E3 +505602.749}
SPL {X  -165.650, Y  +513.685, Z    +0.000, E1   -30.234, E3 +505616.246}
SPL {X  -165.650, Y  +517.919, Z    +0.000, E1   -30.227, E3 +505631.153}
SPL {X  -165.650, Y  +521.521, Z    +0.000, E1   -30.210, E3 +505643.828}
SPL {X  -165.650, Y  +525.344, Z    +0.000, E1   -30.269, E3 +505656.934}
SPL {X  -165.650, Y  +528.152, Z    +0.000, E1   -29.991, E3 +505668.575}
SPL {X  -165.650, Y  +531.783, Z    +0.000, E1   -30.416, E3 +505678.467}
SPL {X  -165.650, Y  +534.115, Z    +0.000, E1   -30.089, E3 +505688.850}
SPL {X  -165.650, Y  +537.522, Z    +0.000, E1   -30.251, E3 +505699.764}
SPL {X  -165.650, Y  +540.621, Z    +0.000, E1   -30.014, E3 +505712.325}
SPL {X  -165.650, Y  +544.944, Z    +0.000, E1   -30.447, E3 +505724.524}
SPL {X  -165.650, Y  +547.199, Z    +0.000, E1   -30.132, E3 +505734.498}
SPL {X  -165.650, Y  +550.512, Z    +0.000, E1   -30.197, E3 +505745.824}
SPL {X  -165.650, Y  +553.852, Z    +0.000, E1   -30.156, E3 +505757.765}
SPL {X  -165.650, Y  +557.277, Z    +0.000, E1   -30.150, E3 +505769.939}
SPL {X  -165.650, Y  +561.168, Z    +0.000, E1   -30.194, E3 +505783.320}
SPL {X  -165.650, Y  +565.528, Z    +0.000, E1   -30.192, E3 +505798.803}
SPL {X  -165.650, Y  +570.048, Z    +0.000, E1   -30.238, E3 +505814.234}
SPL {X  -165.650, Y  +573.110, Z    +0.000, E1   -30.057, E3 +505826.219}
SPL {X  -165.650, Y  +577.587, Z    +0.000, E1   -30.270, E3 +505840.658}
SPL {X  -165.650, Y  +581.190, Z    +0.000, E1   -30.107, E3 +505854.298}
SPL {X  -165.650, Y  +585.053, Z    +0.000, E1   -30.090, E3 +505868.168}
ENDSPLINE

SPLINE
SPL {X  -165.650, Y  +484.445, Z    +0.000, E1   +32.277, E3 +505885.572}
SPL {X  -165.650, Y  +481.524, Z    +0.000, E1   +31.089, E3 +505903.023}
SPL {X  -165.650, Y  +478.014, Z    +0.000, E1   +30.826, E3 +505916.630}
SPL {X  -165.650, Y  +474.473, Z    +0.000, E1   +30.943, E3 +505927.955}
SPL {X  -165.650, Y  +471.826, Z    +0.000, E1   +30.770, E3 +505938.138}
SPL {X  -165.650, Y  +467.753, Z    +0.000, E1   +30.878, E3 +505951.512}
SPL {X  -165.650, Y  +463.837, Z    +0.000, E1   +30.924, E3 +505964.446}
SPL {X  -165.650, Y  +461.106, Z    +0.000, E1   +30.916, E3 +505973.833}
SPL {X  -165.650, Y  +458.435, Z    +0.000, E1   +30.759, E3 +505984.041}
SPL {X  -165.650, Y  +454.220, Z    +0.000, E1   +30.954, E3 +505997.274}
SPL {X  -165.650, Y  +450.433, Z    +0.000, E1   +30.789, E3 +506011.238}
SPL {X  -165.650, Y  +447.097, Z    +0.000, E1   +30.843, E3 +506022.287}
SPL {X  -165.650, Y  +443.673, Z    +0.000, E1   +30.907, E3 +506033.595}
SPL {X  -165.650, Y  +440.976, Z    +0.000, E1   +30.719, E3 +506044.051}
SPL {X  -165.650, Y  +436.324, Z    +0.000, E1   +30.994, E3 +506058.338}
SPL {X  -165.650, Y  +432.765, Z    +0.000, E1   +30.831, E3 +506071.338}
SPL {X  -165.650, Y  +429.309, Z    +0.000, E1   +30.920, E3 +506082.679}
SPL {X  -165.650, Y  +424.918, Z    +0.000, E1   +30.862, E3 +506098.136}
SPL {X  -165.650, Y  +421.437, Z    +0.000, E1   +30.833, E3 +506110.104}
SPL {X  -165.650, Y  +417.366, Z    +0.000, E1   +30.879, E3 +506123.945}
SPL {X  -165.650, Y  +413.181, Z    +0.000, E1   +30.815, E3 +506138.542}
SPL {X  -165.650, Y  +408.547, Z    +0.000, E1   +30.964, E3 +506153.545}
SPL {X  -165.650, Y  +403.421, Z    +0.000, E1   +30.863, E3 +506171.763}
SPL {X  -165.650, Y  +398.147, Z    +0.000, E1   +30.902, E3 +506189.523}
SPL {X  -165.650, Y  +394.694, Z    +0.000, E1   +30.805, E3 +506201.832}
SPL {X  -165.650, Y  +390.331, Z    +0.000, E1   +30.892, E3 +506216.408}
SPL {X  -165.650, Y  +384.849, Z    +0.000, E1   +30.885, E3 +506235.211}
SPL {X  -165.650, Y  +380.752, Z    +0.000, E1   +30.927, E3 +506248.713}
SPL {X  -165.648, Y  +377.739, Z    +0.000, E1   +30.835, E3 +506259.722}
SPL {X  -165.594, Y  +374.183, Z    +0.000, E1   +30.878, E3 +506271.559}
SPL {X  -165.492, Y  +371.263, Z    +0.000, E1   +30.913, E3 +506281.254}
SPL {X  -165.379, Y  +369.027, Z    +0.000, E1   +30.727, E3 +506290.193}
SPL {X  -165.167, Y  +365.866, Z    +0.000, E1   +30.741, E3 +506300.967}
SPL {X  -164.892, Y  +362.671, Z    +0.000, E1   +30.830, E3 +506311.291}
SPL {X  -164.570, Y  +359.612, Z    +0.000, E1   +30.773, E3 +506322.103}
SPL {X  -164.104, Y  +355.923, Z    +0.000, E1   +30.626, E3 +506335.820}
SPL {X  -163.573, Y  +352.353, Z    +0.000, E1   +30.451, E3 +506349.085}
SPL {X  -162.476, Y  +346.230, Z    +0.000, E1   +31.677, E3 +506361.666}
SPL {X  -152.976, Y  +314.952, Z    +0.000, E1   +38.607, E3 +506410.631}
SPL {X  -137.967, Y  +286.821, Z    +0.000, E1   +43.969, E3 +506453.852}
ENDSPLINE

SPLINE
SPL {X  -149.143, Y  +306.414, Z    +0.000, E1   +36.361, E3 +506504.984}
SPL {X  -163.091, Y  +349.496, Z    +0.000, E1   +19.699, E3 +506461.767}
SPL {X  -164.704, Y  +360.824, Z    +0.000, E1   +13.856, E3 +506463.108}
SPL {X  -165.510, Y  +371.680, Z    +0.000, E1    +7.684, E3 +506465.746}
SPL {X  -165.628, Y  +375.818, Z    +0.000, E1    +5.016, E3 +506473.675}
SPL {X  -165.650, Y  +383.362, Z    +0.000, E1    +0.177, E3 +506454.709}
SPL {X  -165.650, Y  +383.923, Z    +0.000, E1    -0.215, E3 +506467.866}
SPL {X  -165.650, Y  +388.083, Z    +0.000, E1    -3.355, E3 +506466.730}
SPL {X  -165.650, Y  +393.983, Z    +0.000, E1    -8.501, E3 +506463.128}
SPL {X  -165.650, Y  +402.241, Z    +0.000, E1   -16.711, E3 +506457.640}
SPL {X  -165.650, Y  +414.811, Z    +0.000, E1   -28.314, E3 +506457.170}
SPL {X  -165.650, Y  +423.479, Z    +0.000, E1   -29.012, E3 +506481.099}
SPL {X  -165.650, Y  +441.276, Z    +0.000, E1   -37.343, E3 +506492.788}
SPL {X  -165.650, Y  +462.890, Z    +0.000, E1   -40.484, E3 +506526.871}
ENDSPLINE

SPLINE
SPL {X  -165.650, Y  +446.920, Z    +0.000, E1   -31.238, E3 +506539.197}
ENDSPLINE

SPLINE
SPL {X  -165.650, Y  +447.935, Z    +0.000, E1   -30.213, E3 +506549.484}
SPL {X  -165.650, Y  +451.020, Z    +0.000, E1   -30.224, E3 +506560.305}
SPL {X  -165.650, Y  +454.519, Z    +0.000, E1   -30.374, E3 +506571.487}
SPL {X  -165.650, Y  +457.429, Z    +0.000, E1   -30.029, E3 +506584.189}
SPL {X  -165.650, Y  +461.678, Z    +0.000, E1   -30.426, E3 +506596.314}
SPL {X  -165.650, Y  +463.853, Z    +0.000, E1   -30.103, E3 +506606.153}
SPL {X  -165.650, Y  +468.397, Z    +0.000, E1   -30.302, E3 +506620.957}
SPL {X  -165.650, Y  +472.566, Z    +0.000, E1   -30.124, E3 +506636.666}
SPL {X  -165.650, Y  +476.540, Z    +0.000, E1   -30.193, E3 +506650.210}
SPL {X  -165.650, Y  +481.042, Z    +0.000, E1   -30.192, E3 +506666.156}
SPL {X  -165.650, Y  +485.236, Z    +0.000, E1   -30.294, E3 +506680.011}
SPL {X  -165.650, Y  +489.057, Z    +0.000, E1   -30.341, E3 +506693.217}
SPL {X  -165.650, Y  +491.647, Z    +0.000, E1   -29.894, E3 +506705.150}
SPL {X  -165.650, Y  +495.051, Z    +0.000, E1   -30.213, E3 +506715.079}
SPL {X  -165.650, Y  +498.418, Z    +0.000, E1   -30.282, E3 +506726.372}
SPL {X  -165.650, Y  +502.421, Z    +0.000, E1   -30.263, E3 +506740.730}
SPL {X  -165.650, Y  +506.344, Z    +0.000, E1   -30.129, E3 +506755.259}
SPL {X  -165.650, Y  +509.866, Z    +0.000, E1   -30.236, E3 +506766.929}
SPL {X  -165.650, Y  +513.685, Z    +0.000, E1   -30.234, E3 +506780.425}
SPL {X  -165.650, Y  +517.919, Z    +0.000, E1   -30.227, E3 +506795.332}
SPL {X  -165.650, Y  +521.521, Z    +0.000, E1   -30.210, E3 +506808.007}
SPL {X  -165.650, Y  +525.344, Z    +0.000, E1   -30.269, E3 +506821.113}
SPL {X  -165.650, Y  +528.152, Z    +0.000, E1   -29.991, E3 +506832.754}
SPL {X  -165.650, Y  +531.783, Z    +0.000, E1   -30.416, E3 +506842.647}
SPL {X  -165.650, Y  +534.115, Z    +0.000, E1   -30.089, E3 +506853.029}
SPL {X  -165.650, Y  +537.522, Z    +0.000, E1   -30.251, E3 +506863.943}
SPL {X  -165.650, Y  +540.621, Z    +0.000, E1   -30.014, E3 +506876.504}
SPL {X  -165.650, Y  +544.944, Z    +0.000, E1   -30.447, E3 +506888.704}
SPL {X  -165.650, Y  +548.549, Z    +0.000, E1   -30.216, E3 +506903.027}
SPL {X  -165.650, Y  +553.092, Z    +0.000, E1   -30.157, E3 +506919.370}
SPL {X  -165.650, Y  +556.274, Z    +0.000, E1   -30.127, E3 +506930.624}
SPL {X  -165.650, Y  +560.243, Z    +0.000, E1   -30.214, E3 +506944.290}
SPL {X  -165.650, Y  +565.528, Z    +0.000, E1   -30.192, E3 +506962.982}
SPL {X  -165.650, Y  +570.048, Z    +0.000, E1   -30.238, E3 +506978.413}
SPL {X  -165.650, Y  +573.110, Z    +0.000, E1   -30.057, E3 +506990.398}
SPL {X  -165.650, Y  +577.587, Z    +0.000, E1   -30.270, E3 +507004.837}
SPL {X  -165.650, Y  +581.190, Z    +0.000, E1   -30.107, E3 +507018.477}
SPL {X  -165.650, Y  +585.053, Z    +0.000, E1   -30.090, E3 +507032.347}
ENDSPLINE

SPLINE
SPL {X  -165.650, Y  +484.445, Z    +0.000, E1   +32.277, E3 +507049.751}
SPL {X  -165.650, Y  +481.524, Z    +0.000, E1   +31.089, E3 +507067.202}
SPL {X  -165.650, Y  +478.014, Z    +0.000, E1   +30.826, E3 +507080.810}
SPL {X  -165.650, Y  +474.473, Z    +0.000, E1   +30.943, E3 +507092.134}
SPL {X  -165.650, Y  +471.826, Z    +0.000, E1   +30.770, E3 +507102.317}
SPL {X  -165.650, Y  +467.753, Z    +0.000, E1   +30.878, E3 +507115.691}
SPL {X  -165.650, Y  +463.837, Z    +0.000, E1   +30.924, E3 +507128.625}
SPL {X  -165.650, Y  +461.106, Z    +0.000, E1   +30.916, E3 +507138.012}
SPL {X  -165.650, Y  +457.156, Z    +0.000, E1   +30.860, E3 +507152.088}
SPL {X  -165.650, Y  +453.156, Z    +0.000, E1   +30.934, E3 +507165.062}
SPL {X  -165.650, Y  +450.433, Z    +0.000, E1   +30.789, E3 +507175.418}
SPL {X  -165.650, Y  +447.097, Z    +0.000, E1   +30.843, E3 +507186.466}
SPL {X  -165.650, Y  +443.673, Z    +0.000, E1   +30.907, E3 +507197.774}
SPL {X  -165.650, Y  +439.486, Z    +0.000, E1   +30.857, E3 +507212.583}
SPL {X  -165.650, Y  +434.043, Z    +0.000, E1   +30.950, E3 +507230.599}
SPL {X  -165.650, Y  +430.419, Z    +0.000, E1   +30.895, E3 +507243.102}
SPL {X  -165.650, Y  +427.340, Z    +0.000, E1   +30.870, E3 +507253.929}
SPL {X  -165.650, Y  +422.641, Z    +0.000, E1   +30.884, E3 +507270.018}
SPL {X  -165.650, Y  +417.366, Z    +0.000, E1   +30.879, E3 +507288.124}
SPL {X  -165.650, Y  +412.139, Z    +0.000, E1   +30.870, E3 +507306.073}
SPL {X  -165.650, Y  +406.834, Z    +0.000, E1   +30.919, E3 +507323.902}
SPL {X  -165.650, Y  +402.516, Z    +0.000, E1   +30.874, E3 +507338.824}
SPL {X  -165.650, Y  +398.147, Z    +0.000, E1   +30.902, E3 +507353.702}
SPL {X  -165.650, Y  +394.694, Z    +0.000, E1   +30.805, E3 +507366.011}
SPL {X  -165.650, Y  +391.522, Z    +0.000, E1   +30.837, E3 +507376.692}
SPL {X  -165.650, Y  +387.533, Z    +0.000, E1   +30.858, E3 +507390.318}
SPL {X  -165.650, Y  +383.627, Z    +0.000, E1   +30.885, E3 +507403.378}
SPL {X  -165.650, Y  +380.752, Z    +0.000, E1   +30.927, E3 +507412.892}
SPL {X  -165.648, Y  +377.739, Z    +0.000, E1   +30.835, E3 +507423.901}
SPL {X  -165.594, Y  +374.183, Z    +0.000, E1   +30.878, E3 +507435.738}
SPL {X  -165.492, Y  +371.263, Z    +0.000, E1   +30.913, E3 +507445.433}
SPL {X  -165.379, Y  +369.027, Z    +0.000, E1   +30.727, E3 +507454.372}
SPL {X  -165.167, Y  +365.866, Z    +0.000, E1   +30.741, E3 +507465.146}
SPL {X  -164.892, Y  +362.671, Z    +0.000, E1   +30.830, E3 +507475.470}
SPL {X  -164.570, Y  +359.612, Z    +0.000, E1   +30.773, E3 +507486.283}
SPL {X  -164.104, Y  +355.923, Z    +0.000, E1   +30.626, E3 +507499.999}
SPL {X  -163.573, Y  +352.353, Z    +0.000, E1   +30.451, E3 +507513.264}
SPL {X  -162.476, Y  +346.230, Z    +0.000, E1   +31.677, E3 +507525.845}
SPL {X  -152.976, Y  +314.952, Z    +0.000, E1   +38.607, E3 +507574.810}
SPL {X  -137.967, Y  +286.821, Z    +0.000, E1   +43.969, E3 +507618.031}
ENDSPLINE

SPLINE
SPL {X  -153.316, Y  +315.777, Z    +0.000, E1   +33.140, E3 +507660.658}
SPL {X  -164.446, Y  +358.564, Z    +0.000, E1   +15.149, E3 +507625.869}
SPL {X  -165.379, Y  +369.025, Z    +0.000, E1    +9.158, E3 +507631.594}
SPL {X  -165.612, Y  +374.969, Z    +0.000, E1    +5.630, E3 +507634.270}
SPL {X  -165.650, Y  +383.362, Z    +0.000, E1    +0.177, E3 +507618.888}
SPL {X  -165.650, Y  +383.923, Z    +0.000, E1    -0.215, E3 +507632.045}
SPL {X  -165.650, Y  +388.083, Z    +0.000, E1    -3.355, E3 +507630.909}
SPL {X  -165.650, Y  +393.983, Z    +0.000, E1    -8.501, E3 +507627.307}
SPL {X  -165.650, Y  +402.241, Z    +0.000, E1   -16.711, E3 +507621.819}
SPL {X  -165.650, Y  +416.345, Z    +0.000, E1   -29.511, E3 +507621.611}
SPL {X  -165.650, Y  +422.331, Z    +0.000, E1   -27.760, E3 +507647.110}
SPL {X  -165.650, Y  +441.276, Z    +0.000, E1   -37.343, E3 +507656.967}
SPL {X  -165.650, Y  +462.890, Z    +0.000, E1   -40.484, E3 +507691.050}
ENDSPLINE

SPLINE
SPL {X  -165.650, Y  +446.920, Z    +0.000, E1   -31.238, E3 +507703.376}
ENDSPLINE

SPLINE
SPL {X  -165.650, Y  +447.935, Z    +0.000, E1   -30.213, E3 +507713.664}
SPL {X  -165.650, Y  +451.020, Z    +0.000, E1   -30.224, E3 +507724.484}
SPL {X  -165.650, Y  +454.519, Z    +0.000, E1   -30.374, E3 +507735.666}
SPL {X  -165.650, Y  +457.429, Z    +0.000, E1   -30.029, E3 +507748.368}
SPL {X  -165.650, Y  +461.678, Z    +0.000, E1   -30.426, E3 +507760.493}
SPL {X  -165.650, Y  +463.853, Z    +0.000, E1   -30.103, E3 +507770.332}
SPL {X  -165.650, Y  +468.397, Z    +0.000, E1   -30.302, E3 +507785.136}
SPL {X  -165.650, Y  +472.566, Z    +0.000, E1   -30.124, E3 +507800.845}
SPL {X  -165.650, Y  +476.540, Z    +0.000, E1   -30.193, E3 +507814.390}
SPL {X  -165.650, Y  +481.042, Z    +0.000, E1   -30.192, E3 +507830.335}
SPL {X  -165.650, Y  +485.236, Z    +0.000, E1   -30.294, E3 +507844.190}
SPL {X  -165.650, Y  +489.057, Z    +0.000, E1   -30.341, E3 +507857.396}
SPL {X  -165.650, Y  +491.647, Z    +0.000, E1   -29.894, E3 +507869.330}
SPL {X  -165.650, Y  +495.051, Z    +0.000, E1   -30.213, E3 +507879.258}
SPL {X  -165.650, Y  +498.418, Z    +0.000, E1   -30.282, E3 +507890.551}
SPL {X  -165.650, Y  +502.421, Z    +0.000, E1   -30.263, E3 +507904.909}
SPL {X  -165.650, Y  +506.344, Z    +0.000, E1   -30.129, E3 +507919.438}
SPL {X  -165.650, Y  +509.866, Z    +0.000, E1   -30.236, E3 +507931.108}
SPL {X  -165.650, Y  +513.685, Z    +0.000, E1   -30.234, E3 +507944.604}
SPL {X  -165.650, Y  +517.919, Z    +0.000, E1   -30.227, E3 +507959.511}
SPL {X  -165.650, Y  +521.521, Z    +0.000, E1   -30.210, E3 +507972.186}
SPL {X  -165.650, Y  +525.344, Z    +0.000, E1   -30.269, E3 +507985.292}
SPL {X  -165.650, Y  +528.152, Z    +0.000, E1   -29.991, E3 +507996.933}
SPL {X  -165.650, Y  +531.783, Z    +0.000, E1   -30.416, E3 +508006.826}
SPL {X  -165.650, Y  +534.115, Z    +0.000, E1   -30.089, E3 +508017.208}
SPL {X  -165.650, Y  +537.522, Z    +0.000, E1   -30.251, E3 +508028.122}
SPL {X  -165.650, Y  +540.621, Z    +0.000, E1   -30.014, E3 +508040.683}
SPL {X  -165.650, Y  +544.944, Z    +0.000, E1   -30.447, E3 +508052.883}
SPL {X  -165.650, Y  +548.549, Z    +0.000, E1   -30.216, E3 +508067.206}
SPL {X  -165.650, Y  +553.092, Z    +0.000, E1   -30.157, E3 +508083.549}
SPL {X  -165.650, Y  +556.274, Z    +0.000, E1   -30.127, E3 +508094.803}
SPL {X  -165.650, Y  +560.243, Z    +0.000, E1   -30.214, E3 +508108.469}
SPL {X  -165.650, Y  +565.528, Z    +0.000, E1   -30.192, E3 +508127.161}
SPL {X  -165.650, Y  +570.048, Z    +0.000, E1   -30.238, E3 +508142.593}
SPL {X  -165.650, Y  +573.110, Z    +0.000, E1   -30.057, E3 +508154.578}
SPL {X  -165.650, Y  +577.587, Z    +0.000, E1   -30.270, E3 +508169.017}
SPL {X  -165.650, Y  +581.190, Z    +0.000, E1   -30.107, E3 +508182.656}
SPL {X  -165.650, Y  +585.053, Z    +0.000, E1   -30.090, E3 +508196.526}
ENDSPLINE

SPLINE
SPL {X  -165.650, Y  +484.445, Z    +0.000, E1   +32.277, E3 +508213.931}
SPL {X  -165.650, Y  +481.524, Z    +0.000, E1   +31.089, E3 +508231.381}
SPL {X  -165.650, Y  +478.014, Z    +0.000, E1   +30.826, E3 +508244.989}
SPL {X  -165.650, Y  +474.473, Z    +0.000, E1   +30.943, E3 +508256.313}
SPL {X  -165.650, Y  +471.826, Z    +0.000, E1   +30.770, E3 +508266.497}
SPL {X  -165.650, Y  +467.753, Z    +0.000, E1   +30.878, E3 +508279.870}
SPL {X  -165.650, Y  +463.837, Z    +0.000, E1   +30.924, E3 +508292.804}
SPL {X  -165.650, Y  +461.106, Z    +0.000, E1   +30.916, E3 +508302.191}
SPL {X  -165.650, Y  +457.156, Z    +0.000, E1   +30.860, E3 +508316.267}
SPL {X  -165.650, Y  +453.156, Z    +0.000, E1   +30.934, E3 +508329.241}
SPL {X  -165.650, Y  +450.433, Z    +0.000, E1   +30.789, E3 +508339.597}
SPL {X  -165.650, Y  +447.097, Z    +0.000, E1   +30.843, E3 +508350.645}
SPL {X  -165.650, Y  +443.673, Z    +0.000, E1   +30.907, E3 +508361.953}
SPL {X  -165.650, Y  +439.486, Z    +0.000, E1   +30.857, E3 +508376.762}
SPL {X  -165.650, Y  +434.043, Z    +0.000, E1   +30.950, E3 +508394.778}
SPL {X  -165.650, Y  +430.419, Z    +0.000, E1   +30.895, E3 +508407.281}
SPL {X  -165.650, Y  +427.340, Z    +0.000, E1   +30.870, E3 +508418.108}
SPL {X  -165.650, Y  +422.641, Z    +0.000, E1   +30.884, E3 +508434.197}
SPL {X  -165.650, Y  +418.489, Z    +0.000, E1   +30.835, E3 +508448.579}
SPL {X  -165.650, Y  +414.127, Z    +0.000, E1   +30.869, E3 +508463.488}
SPL {X  -165.650, Y  +408.547, Z    +0.000, E1   +30.964, E3 +508481.903}
SPL {X  -165.650, Y  +405.433, Z    +0.000, E1   +30.730, E3 +508493.880}
SPL {X  -165.650, Y  +401.473, Z    +0.000, E1   +30.933, E3 +508506.329}
SPL {X  -165.650, Y  +396.018, Z    +0.000, E1   +30.861, E3 +508525.514}
SPL {X  -165.650, Y  +390.331, Z    +0.000, E1   +30.892, E3 +508544.766}
SPL {X  -165.650, Y  +384.849, Z    +0.000, E1   +30.885, E3 +508563.569}
SPL {X  -165.650, Y  +380.752, Z    +0.000, E1   +30.927, E3 +508577.071}
SPL {X  -165.648, Y  +377.739, Z    +0.000, E1   +30.835, E3 +508588.081}
SPL {X  -165.594, Y  +374.183, Z    +0.000, E1   +30.878, E3 +508599.917}
SPL {X  -165.492, Y  +371.263, Z    +0.000, E1   +30.913, E3 +508609.612}
SPL {X  -165.379, Y  +369.027, Z    +0.000, E1   +30.727, E3 +508618.551}
SPL {X  -165.167, Y  +365.866, Z    +0.000, E1   +30.741, E3 +508629.325}
SPL {X  -164.892, Y  +362.671, Z    +0.000, E1   +30.830, E3 +508639.649}
SPL {X  -164.570, Y  +359.612, Z    +0.000, E1   +30.773, E3 +508650.462}
SPL {X  -164.104, Y  +355.923, Z    +0.000, E1   +30.626, E3 +508664.178}
SPL {X  -163.573, Y  +352.353, Z    +0.000, E1   +30.451, E3 +508677.443}
SPL {X  -162.476, Y  +346.230, Z    +0.000, E1   +31.677, E3 +508690.024}
SPL {X  -152.976, Y  +314.952, Z    +0.000, E1   +38.607, E3 +508738.989}
SPL {X  -137.967, Y  +286.821, Z    +0.000, E1   +43.969, E3 +508782.210}
ENDSPLINE

SPLINE
SPL {X  -153.316, Y  +315.777, Z    +0.000, E1   +33.140, E3 +508824.838}
SPL {X  -164.446, Y  +358.564, Z    +0.000, E1   +15.149, E3 +508790.048}
SPL {X  -165.510, Y  +371.680, Z    +0.000, E1    +7.684, E3 +508794.104}
SPL {X  -165.628, Y  +375.818, Z    +0.000, E1    +5.016, E3 +508802.033}
SPL {X  -165.650, Y  +383.362, Z    +0.000, E1    +0.177, E3 +508783.067}
SPL {X  -165.650, Y  +383.923, Z    +0.000, E1    -0.215, E3 +508796.224}
SPL {X  -165.650, Y  +388.083, Z    +0.000, E1    -3.355, E3 +508795.088}
SPL {X  -165.650, Y  +393.983, Z    +0.000, E1    -8.501, E3 +508791.486}
SPL {X  -165.650, Y  +402.241, Z    +0.000, E1   -16.711, E3 +508785.998}
SPL {X  -165.650, Y  +416.345, Z    +0.000, E1   -29.511, E3 +508785.790}
SPL {X  -165.650, Y  +422.331, Z    +0.000, E1   -27.760, E3 +508811.289}
SPL {X  -165.650, Y  +441.276, Z    +0.000, E1   -37.343, E3 +508821.146}
SPL {X  -165.650, Y  +462.890, Z    +0.000, E1   -40.484, E3 +508855.229}
ENDSPLINE

SPLINE
SPL {X  -165.650, Y  +446.920, Z    +0.000, E1   -31.238, E3 +508867.555}
ENDSPLINE

SPLINE
SPL {X  -165.650, Y  +447.935, Z    +0.000, E1   -30.213, E3 +508877.843}
SPL {X  -165.650, Y  +451.020, Z    +0.000, E1   -30.224, E3 +508888.663}
SPL {X  -165.650, Y  +454.519, Z    +0.000, E1   -30.374, E3 +508899.845}
SPL {X  -165.650, Y  +456.542, Z    +0.000, E1   -29.986, E3 +508909.590}
SPL {X  -165.650, Y  +460.618, Z    +0.000, E1   -30.298, E3 +508921.911}
SPL {X  -165.650, Y  +463.853, Z    +0.000, E1   -30.103, E3 +508934.511}
SPL {X  -165.650, Y  +467.246, Z    +0.000, E1   -30.279, E3 +508945.242}
SPL {X  -165.650, Y  +469.780, Z    +0.000, E1   -30.237, E3 +508954.367}
SPL {X  -165.650, Y  +472.566, Z    +0.000, E1   -30.124, E3 +508965.025}
SPL {X  -165.650, Y  +476.540, Z    +0.000, E1   -30.193, E3 +508978.569}
SPL {X  -165.650, Y  +480.320, Z    +0.000, E1   -30.163, E3 +508992.046}
SPL {X  -165.650, Y  +484.477, Z    +0.000, E1   -30.274, E3 +509005.936}
SPL {X  -165.650, Y  +488.041, Z    +0.000, E1   -30.253, E3 +509018.491}
SPL {X  -165.650, Y  +491.281, Z    +0.000, E1   -30.148, E3 +509030.629}
SPL {X  -165.650, Y  +495.051, Z    +0.000, E1   -30.213, E3 +509043.438}
SPL {X  -165.650, Y  +498.418, Z    +0.000, E1   -30.282, E3 +509054.730}
SPL {X  -165.650, Y  +502.421, Z    +0.000, E1   -30.263, E3 +509069.088}
SPL {X  -165.650, Y  +506.344, Z    +0.000, E1   -30.129, E3 +509083.617}
SPL {X  -165.650, Y  +509.866, Z    +0.000, E1   -30.236, E3 +509095.287}
SPL {X  -165.650, Y  +513.685, Z    +0.000, E1   -30.234, E3 +509108.783}
SPL {X  -165.650, Y  +517.104, Z    +0.000, E1   -30.280, E3 +509120.335}
SPL {X  -165.650, Y  +520.621, Z    +0.000, E1   -30.198, E3 +509133.414}
SPL {X  -165.650, Y  +525.344, Z    +0.000, E1   -30.269, E3 +509149.471}
SPL {X  -165.650, Y  +528.152, Z    +0.000, E1   -29.991, E3 +509161.112}
SPL {X  -165.650, Y  +531.783, Z    +0.000, E1   -30.416, E3 +509171.005}
SPL {X  -165.650, Y  +534.115, Z    +0.000, E1   -30.089, E3 +509181.387}
SPL {X  -165.650, Y  +537.522, Z    +0.000, E1   -30.251, E3 +509192.301}
SPL {X  -165.650, Y  +540.621, Z    +0.000, E1   -30.014, E3 +509204.862}
SPL {X  -165.650, Y  +544.944, Z    +0.000, E1   -30.447, E3 +509217.062}
SPL {X  -165.650, Y  +547.199, Z    +0.000, E1   -30.132, E3 +509227.035}
SPL {X  -165.650, Y  +550.512, Z    +0.000, E1   -30.197, E3 +509238.361}
SPL {X  -165.650, Y  +553.852, Z    +0.000, E1   -30.156, E3 +509250.302}
SPL {X  -165.650, Y  +557.277, Z    +0.000, E1   -30.150, E3 +509262.476}
SPL {X  -165.650, Y  +561.168, Z    +0.000, E1   -30.194, E3 +509275.858}
SPL {X  -165.650, Y  +565.528, Z    +0.000, E1   -30.192, E3 +509291.341}
SPL {X  -165.650, Y  +570.048, Z    +0.000, E1   -30.238, E3 +509306.772}
SPL {X  -165.650, Y  +573.110, Z    +0.000, E1   -30.057, E3 +509318.757}
SPL {X  -165.650, Y  +577.587, Z    +0.000, E1   -30.270, E3 +509333.196}
SPL {X  -165.650, Y  +581.190, Z    +0.000, E1   -30.107, E3 +509346.835}
SPL {X  -165.650, Y  +585.053, Z    +0.000, E1   -30.090, E3 +509360.705}
ENDSPLINE

SPLINE
SPL {X  -165.650, Y  +484.968, Z    +0.000, E1   +32.508, E3 +509374.671}
SPL {X  -165.650, Y  +482.515, Z    +0.000, E1   +31.539, E3 +509389.199}
ENDSPLINE

SLIN {X  -200.000, Y  +530.000, E1    +0.000}
HALT
END
